PROGRAM HMI_Crush_Indicator
VAR
	dwCrushFlag: DWORD;
	bCrushFlag: BOOL;
END_VAR

IF GV_LIFT.CRUSH_PROTECTION_INDICATOR_IN THEN
	dwCrushFlag := GV_HMI.dwGreen;
	bCrushFlag := FALSE;
ELSE dwCrushFlag := GV_HMI.dwRed;
	bCrushFlag := TRUE;
END_IF

END_PROGRAM

(* stored: Version 1.1.0.1, ProductVersion 3.1.4022.12
   POU HMI_Crush_Indicator: Id {2a3636d1-b05b-4fb3-9c6d-842facab1bce}, SpecialFunc None *)
